(* IEC 61131-3 sources: CodesysTest/export/SX_1195.dev/Plc Logic/Application/PRJ Specific/Motion/Motors/Oriental AZD/AZD4A-KED/FB_AZDKABase.pou/TargetPositionInSteps.prop, 1 file *)

(* ---- Get.pm.st ---- *)
(*#-#-#-#-#-#-#-#-#-#---Declaration---#-#-#-#-#-#-#-#-#-#-#-#-#*)

VAR
END_VAR
(*#-#-#-#-#-#-#-#-#-#---Implementation---#-#-#-#-#-#-#-#-#-#-#-#-#*)

TargetPositionInSteps := (targetPosDist - zeroOffset) * TO_REAL(axisData.config.stepsPerInch);
IF axisData.config.reversePolarity THEN
	TargetPositionInSteps := TargetPositionInSteps * -1;
END_IF
